// TwinCAT 3 PLC project Test_Proj
// ProgramVersion: 3.1.4026.14
// libraries:
//   Base Library, * (Beckhoff UK)
//   Tc3PlcTestSuite, * (Simmel)
//   [Runner Library], * (Beckhoff UK)
// project tree:
//   / PlcTask.TcTTO
//   POUs/ MAIN.TcPOU, MockObj.TcPOU, RunnerTestSuite.TcPOU
// real-time tasks:
//   TASK PlcTask: cycle T#10ms, priority 20, ADS port 350

CONFIGURATION Test_Proj
    RESOURCE PLC ON TwinCAT3
        TASK PlcTask(INTERVAL := T#10ms, PRIORITY := 20);
        PROGRAM MAIN WITH PlcTask : MAIN;
    END_RESOURCE
END_CONFIGURATION

// ---- POUs/MAIN.TcPOU
PROGRAM MAIN
VAR
	ObjRunnerTestSuite : RunnerTestSuite;
END_VAR

ObjRunnerTestSuite();

END_PROGRAM

// ---- POUs/RunnerTestSuite.TcPOU
FUNCTION_BLOCK RunnerTestSuite
VAR
	TestObjRunner : ObjectRunner;
	ReRun : BOOL;
END_VAR

RejectInvalidInterface_Test();
IncrementObjectCountWhenAdded_Test();
IncrementInitObjCountWhenAdded_Test();
RejectAddingSameModule_Test();
RejectInitCallWithNoModules_Test();
ConfirmInitModulesComplete_Test();
ConfirmRunnerCanDeregAllModules_Test();
RunnerAcceptsModule_Test();
IF ReRun THEN
	TestSuite.ReRunTests();
	ReRun := FALSE;
END_IF

METHOD ConfirmInitModulesComplete_Test : BOOL
VAR_INST
	Expected : BOOL;
	Actual	 : BOOL;
END_VAR
VAR
	TestMockObj : MockObj;
END_VAR
IF TestSuite.Test(__POUNAME()).ExecuteTest() THEN
	Expected := TRUE;
	TestObjRunner.RegisterModule(TestMockObj);
	TestObjRunner.Initialise();
	Actual := TestObjRunner.AreAllModuleInitialised();
	TestObjRunner.DeregisterAllModules();
	TestSuite.Test(__POUNAME()).AssertEqual(Expected, Actual);
END_IF
END_METHOD

METHOD ConfirmRunnerCanDeregAllModules_Test : BOOL
VAR_INST
	Expected : INT;
	Actual	 : INT;
END_VAR
VAR
	TestMockObj1 : MockObj;
	TestMockObj2 : MockObj;
END_VAR
IF TestSuite.Test(__POUNAME()).ExecuteTest() THEN
	Expected := 0;
	TestObjRunner.RegisterModule(TestMockObj1);
	TestObjRunner.RegisterModule(TestMockObj2);
	Actual := TestObjRunner.GetCyclicModuleCount();
	TestObjRunner.DeregisterAllModules();
	Actual := TestObjRunner.GetCyclicModuleCount();
	TestSuite.Test(__POUNAME()).AssertEqual(Expected, Actual);
END_IF
END_METHOD

METHOD IncrementInitObjCountWhenAdded_Test : BOOL
VAR_INST
	Expected : INT := 1;
	Actual	 : INT;
END_VAR
VAR
	TestMockObj : MockObj;
END_VAR
IF TestSuite.Test(__POUNAME()).ExecuteTest() THEN
	TestObjRunner.RegisterModule(TestMockObj);
	Actual := TestObjRunner.GetInitModuleCount();
	TestSuite.Test(__POUNAME()).AssertEqual(Expected, Actual);
	TestObjRunner.DeregisterAllModules();
END_IF
END_METHOD

METHOD IncrementObjectCountWhenAdded_Test : BOOL
VAR_INST
	Expected : INT := 1;
	Actual	 : INT;
END_VAR
VAR
	TestMockObj : MockObj;
END_VAR
IF TestSuite.Test(__POUNAME()).ExecuteTest() THEN
	TestObjRunner.RegisterModule(TestMockObj);
	Actual := TestObjRunner.GetCyclicModuleCount();
	TestSuite.Test(__POUNAME()).AssertEqual(Expected, Actual);
	TestObjRunner.DeregisterAllModules();
END_IF
END_METHOD

METHOD RejectAddingSameModule_Test : BOOL
VAR_INST
	Expected : BOOL := TRUE;
	Actual	 : BOOL;
END_VAR
VAR
	TestMockObj : MockObj;
END_VAR
IF TestSuite.Test(__POUNAME()).ExecuteTest() THEN
	TestObjRunner.RegisterModule(TestMockObj);
	TestObjRunner.RegisterModule(TestMockObj);
	Actual := TestMockObj.IsRegistered();
	TestSuite.Test(__POUNAME()).AssertEqual(Expected, Actual);
	TestObjRunner.DeregisterAllModules();
END_IF
END_METHOD

METHOD RejectInitCallWithNoModules_Test : BOOL
VAR_INST
	Expected : HRESULT;
	Actual	 : HRESULT;
END_VAR
IF TestSuite.Test(__POUNAME()).ExecuteTest() THEN
	Expected := S_False;
	Actual := TestObjRunner.Initialise();
	TestSuite.Test(__POUNAME()).AssertEqual(Expected, Actual);
	TestObjRunner.DeregisterAllModules();
END_IF
END_METHOD

METHOD RejectInvalidInterface_Test : BOOL
VAR_INST
	Expected : HRESULT := -1;
	Actual	 : HRESULT;
END_VAR
IF TestSuite.Test(__POUNAME()).ExecuteTest() THEN
	Actual := TestObjRunner.RegisterModule(16#0);
	TestSuite.Test(__POUNAME()).AssertEqual(Expected, Actual);
END_IF
END_METHOD

METHOD RunnerAcceptsModule_Test : BOOL
VAR_INST
	Expected : BOOL := TRUE;
	Actual	 : BOOL;
END_VAR
VAR
	TestMockObj : MockObj;
END_VAR
IF TestSuite.Test(__POUNAME()).ExecuteTest() THEN
	Actual := SuCCEEDED(TestObjRunner.RegisterModule(TestMockObj));
	TestSuite.Test(__POUNAME()).AssertEqual(Expected, Actual);
	TestObjRunner.DeregisterAllModules();
END_IF
END_METHOD

END_FUNCTION_BLOCK

// ---- POUs/MockObj.TcPOU
FUNCTION_BLOCK MockObj IMPLEMENTS I_Cyclic, I_Initialisable, I_Object, I_Resettable
VAR
	_isRegistered : BOOL;
END_VAR

METHOD Cycle : HRESULT
END_METHOD

METHOD Initialise : HRESULT
END_METHOD

METHOD IsRegistered : BOOL
VAR_INPUT
END_VAR
IsRegistered := _isRegistered;
END_METHOD

METHOD RegisterWithParent
VAR_INPUT
	Runner	: I_HostObjects;
END_VAR
IF NOT _isRegistered THEN
	IF SUCCEEDED( Runner.RegisterCyclic(THIS^)) AND SUCCEEDED(Runner.RegisterInitialise(THIS^)) THEN
		_isRegistered := TRUE;
	ELSE
		_isRegistered := FALSE;
	END_IF
END_IF
END_METHOD

METHOD Reset : Base_Library.HRESULT
END_METHOD

END_FUNCTION_BLOCK
